// TIA Portal V20 export
// export: Created 2025-12-01T14:57:12.0152135Z, ExportSetting None, DisplayName Totally Integrated Automation Portal, DisplayVersion V20 Update 3, DisplayName TIA Portal Openness, DisplayVersion V20 Update 3, DisplayName TIA Portal Version Control Interface, DisplayVersion V20 Update 3, DisplayName STEP 7 Professional, DisplayVersion V20 Update 3, DisplayName STEP 7 Safety, DisplayVersion V20 Update 2, DisplayName WinCC Basic/Comfort/Advanced, DisplayVersion V20 Update 3, DisplayName WinCC Professional, DisplayVersion V20 Update 3, DisplayName WinCC Unified, DisplayVersion V20 Update 3
FUNCTION "FC814_EventosRec_Reset" : Void   // FC814, LAD
{ S7_Optimized_Access := 'FALSE' }
// stored: AutoNumber false, SetENOAutomatically false
   VAR_INPUT
      NumJdT : UInt;   // Numero de JdT recibido el Evento
   END_VAR
   VAR_IN_OUT
      P_Eventos : DWord;   // Puntero al DB de Eventos Recibidos
   END_VAR
   VAR_TEMP
      VarEmisionEvento : Struct
         P_Eventos : DWord;
         DBEventos : Word;
         NumDBEventos : UInt;
         MaxBytes : UInt;
         NumBytes : UInt;
         Valor : UDInt;
         Offset : UInt;
      END_STRUCT;
      DBEventosRec : Word;   // DB de Eventos Recibidos
      VarTempReset : Struct
         Mesa : UInt;
         Mckey : UDInt;
         NumeroUT : UInt;
      END_STRUCT;
      AtributosDeReset : Struct
         Tipo : DWord;
         Operacion : DWord;
         Numero : UDInt;
      END_STRUCT;
      Evento : DWord;   // Etiqueta - Evento
      Atributo : DWord;   // Etiqueta - Atributo
      EtiquetaAtributo : DWord;   // Etiqueta - Conversion de Atributo
      NumeroEvento : UInt;   // Numero de Evento
      NumeroAtributo : UInt;   // Numero de Atributo
      Indice : UInt;
      Leido : UInt;
      OffsetInicial : UInt;
      ValorDeAtributo : UDInt;   // Valor del Atributo
      ReturnValor : Int;
      Cero : Byte;
   END_VAR
BEGIN

NETWORK
TITLE = Inicializar
///////////////////////////////////////////////////////////////////////////////////////////
///////////////////////////////////////////////////////////////////////////////////////////
///////////////////////////////////////////////////////////////////////////////////////////
/// Datos del DB de Recepcion de los Eventos
      L     "JDT1_NDB_EventosRec";  // Cogemos el DB de Eventos Recibidos
      T     #DBEventosRec;
      L     "JDT1_NDB_EventosEmi";
      T     #VarEmisionEvento.DBEventos;
      T     #VarEmisionEvento.NumDBEventos;
      L     "JDT1_MaxBytes";
      T     #VarEmisionEvento.MaxBytes;

/// --- Comprobar que JDT a enviado el Evento

      L     #NumJdT;
      L     2;
      <>I;
      JC    NoRecibido_JdT02;

      L     "JDT2_NDB_EventosRec";  // Cogemos el DB de Eventos Recibidos
      T     #DBEventosRec;
      L     "JDT2_NDB_EventosEmi";
      T     #VarEmisionEvento.DBEventos;
      T     #VarEmisionEvento.NumDBEventos;
      L     "JDT2_MaxBytes";
      T     #VarEmisionEvento.MaxBytes;

NoRecibido_JdT02:NOP   0;



NETWORK
TITLE = Distribucion de los Eventos (LIsta del DB de Conversion)
/////////////////////////////////////////////////////////////////////////
/////////////////////////////////////////////////////////////////////////
/////////////////////////////////////////////////////////////////////////
// Hay que recoger el Evento, para despues repartir
// Despues '{' va el tipo de eventos (2 Bytes)
      L     #P_Eventos;  // Recogo por donde va empieza el evento
      LAR2;  // del Quimarox

      OPN   DB [#DBEventosRec];
      L     DBD [AR2, P#0.0];  // Recogo el tipo de Evento (4 Caracteres)
      T     #Evento;


/////////////////////////////////////////////////////////////////////////
/////////////////////////////////////////////////////////////////////////
/////////////////////////////////////////////////////////////////////////
// Buscar numero de evento
      L     1;
      T     #NumeroEvento;
BucleDeBusqueda_NumeroDeEvento:NOP   0;

// -- Se ha encontrado el Evento Recibido
      L     "DB870_ConversorEventos".EventosRecibidos[#NumeroEvento];
      L     #Evento;
      ==D;
      JC    Encontrado_NumeroDeEvento;

// -- Final de la lista de Eventos Recibidos - No Encontrado
      L     "DB870_ConversorEventos".EventosRecibidos[#NumeroEvento];
      L     0;
      ==D;
      JC    NoEncontrado_NumeroDeEvento;

// --- Maximo del Array de la Lista de Eventos Recibidos - No Encontrado
      L     #NumeroEvento;
      L     "CTE_MaxArrayConversion";
      >=I;
      JC    NoEncontrado_NumeroDeEvento;

// --- Continuar la Busqueda
      L     #NumeroEvento;
      L     1;
      +I;
      T     #NumeroEvento;
      JU    BucleDeBusqueda_NumeroDeEvento;


/////////////////////////////////////////////////////////////////////////
// No es ninguno de los eventos previstos, se pasa a buscar el siguiente
NoEncontrado_NumeroDeEvento:NOP   0;
      TAR2;  // Devuelve por donde va empieza el evento
      T     #P_Eventos;  // del Quimarox
      JU    Final_ListaEventos;



NETWORK
TITLE = ----
/////////////////////////////////////////////////////////////////////////
/////////////////////////////////////////////////////////////////////////
/////////////////////////////////////////////////////////////////////////
// Distribuir dependiendo del Resultado de la Busqueda del Evento Recibido
// Para recoger los Atributos
Encontrado_NumeroDeEvento:NOP   0;
      L     #NumeroEvento;
      JL    NoExiste_NumeroDeEvento;

      JU    NoExiste_NumeroDeEvento;
      JU    NoExiste_NumeroDeEvento;  // Evento (01) - CREA
      JU    NoExiste_NumeroDeEvento;  // Evento (02) - RUTA
      JU    NoExiste_NumeroDeEvento;  // Evento (03) - DRUT
      JU    NoExiste_NumeroDeEvento;  // Evento (04) - RETI
      JU    NoExiste_NumeroDeEvento;  // Evento (05) - BORR
      JU    NoExiste_NumeroDeEvento;  // Evento (06) - DATA
      JU    NoExiste_NumeroDeEvento;  // Evento (07) - ?UT?
      JU    NoExiste_NumeroDeEvento;  // Evento (08) - MOVE
      JU    NoExiste_NumeroDeEvento;  // Evento (09) - DEMB

      JU    NoExiste_NumeroDeEvento;  // Evento (10) - CSTA
      JU    NoExiste_NumeroDeEvento;  // Evento (11) - DIDO

      JU    NoExiste_NumeroDeEvento;  // Evento (12) - ORDE
      JU    NoExiste_NumeroDeEvento;  // Evento (13) - BOET
      JU    NoExiste_NumeroDeEvento;  // Evento (14) - BOBD
      JU    NoExiste_NumeroDeEvento;  // Evento (15) - RUET
      JU    NoExiste_NumeroDeEvento;  // Evento (16) - RUES
      JU    NoExiste_NumeroDeEvento;  // Evento (17) - INIR
      JU    NoExiste_NumeroDeEvento;  // Evento (18) - ?ST?

      JU    NoExiste_NumeroDeEvento;  // Evento (19) - QCRE
      JU    NoExiste_NumeroDeEvento;  // Evento (20) - QPR?

      JU    Atributos_EventosDeReset;  // Evento (21) - CHEA

/////////////////////////////////////////////////////////////////////////
NoExiste_NumeroDeEvento:NOP   0;
      TAR2;  // Devuelve por donde va empieza el evento
      T     #P_Eventos;  // del Router
      JU    Final_ListaEventos;



NETWORK
TITLE = ////////////////////////////////////////////////////////////////////////////////////////////////////////////

NETWORK
TITLE = Analizar la lista de los Atributos del Reset
Atributos_EventosDeReset:NOP   0;

/////////////////////////////////////////////////////////////////////////
/////////////////////////////////////////////////////////////////////////
/////////////////////////////////////////////////////////////////////////
// Inicializa variables de los Atributos de Quimarox
      L     0;
      T     #Cero;

      CALL  FILL
      ( BVAL    := #Cero,
        RET_VAL := #ReturnValor,
        BLK     := #AtributosDeReset
      );  // Inicializa Atributos



NETWORK
TITLE = ----
/////////////////////////////////////////////////////////////////////////
/////////////////////////////////////////////////////////////////////////
// Buscando Atributos o Final del Evento
      +AR2  P#4.0;  // Prepara Puntero para ver los atributos

InicioBucleAtributos_EventosDeReset:NOP   0;
      OPN   DB [#DBEventosRec];
      L     DBB [AR2, P#0.0];
      T     #Leido;

// Inicio de atributo - Ir a tratar los atributos
      L     #Leido;
      L     '[';  // '[' - Inicio de Atributo
      ==I;  // Atributo del Evento
      JC    EncontradoAtributos_EventosDeReset;

// Fin del Evento
      L     #Leido;
      L     '}';  // '}' - Fin del Evento
      ==I;  // Se acabo el evento
      JC    FinalAtributos_EventosDeReset;


// Sin Mensaje
      L     #Leido;
      L     0;  // No hay mas Mensaje
      ==I;  // Se acabo el evento
      JC    FinalAtributos_EventosDeReset;

      +AR2  P#1.0;  // Seguir buscado atributo
      JU    InicioBucleAtributos_EventosDeReset;


/////////////////////////////////////////////////////////////////////////
/////////////////////////////////////////////////////////////////////////
// Se acaba el Evento - Ir a guardar datos del Evento
FinalAtributos_EventosDeReset:NOP   0;
      TAR2;
      T     #P_Eventos;  // Guardo Por donde voy en la lista de eventos
      JU    GuardarDatos_EventosRecibidos;



NETWORK
TITLE = Distribucion de los Atributos del Quimarox (LIsta del DB de Conversion)
EncontradoAtributos_EventosDeReset:NOP   0;

/////////////////////////////////////////////////////////////////////////
/////////////////////////////////////////////////////////////////////////
/////////////////////////////////////////////////////////////////////////
/////////////////////////////////////////////////////////////////////////
// Mirar que Atributo del Evento  es ?
      +AR2  P#1.0;
      OPN   DB [#DBEventosRec];
      L     DBD [AR2, P#0.0];  // Atributo - 4 Caracteres
      T     #Atributo;

/////////////////////////////////////////////////////////////////////////
/////////////////////////////////////////////////////////////////////////
/////////////////////////////////////////////////////////////////////////
// Buscar numero de Atributo
      L     1;
      T     #NumeroAtributo;
BucleDeBusqueda_NumeroDeAtributoDeReset:NOP   0;

// -- Se ha encontrado el Atributo Recibido
      L     "DB870_ConversorEventos".AtributosRecibidosDeReset[#NumeroAtributo];
      L     #Atributo;
      ==D;
      JC    Encontrado_NumeroDeAtributoDeReset;

// -- Final de la lista de Atributo Recibidos - No Encontrado
      L     "DB870_ConversorEventos".AtributosRecibidosDeReset[#NumeroAtributo];
      L     0;
      ==D;
      JC    InicioBucleAtributos_EventosDeReset;

// --- Maximo del Array de la Lista de Atributo Recibidos - No Encontrado
      L     #NumeroAtributo;
      L     "CTE_MaxArrayConversion";
      >=I;
      JC    InicioBucleAtributos_EventosDeReset;


// --- Continuar la Busqueda
      L     #NumeroAtributo;
      L     1;
      +I;
      T     #NumeroAtributo;
      JU    BucleDeBusqueda_NumeroDeAtributoDeReset;



NETWORK
TITLE = ----
/////////////////////////////////////////////////////////////////////////
/////////////////////////////////////////////////////////////////////////
/////////////////////////////////////////////////////////////////////////
// Distribuir dependiendo del Resultado de la Busqueda de Atributo Recibido
Encontrado_NumeroDeAtributoDeReset:NOP   0;
      L     #NumeroAtributo;
      JL    NoExiste_NumeroDeAtibutoDeReset;

      JU    NoExiste_NumeroDeAtibutoDeReset;
      JU    AtributoDeReset_TIPO;  // Atributo (01) - TIPO
      JU    AtributoDeReset_NUME;  // Atributo (02) - NUME
      JU    AtributoDeReset_OPER;  // Atributo (03) - OPER


/////////////////////////////////////////////////////////////////////////
NoExiste_NumeroDeAtibutoDeReset:NOP   0;
      JU    InicioBucleAtributos_EventosDeReset;



NETWORK
TITLE = ---- ---- Recoger el Atributo de Quimarox - TIPO
/////////////////////////////////////////////////////////////////////////
/////////////////////////////////////////////////////////////////////////
/////////////////////////////////////////////////////////////////////////
AtributoDeReset_TIPO:NOP   0;
      +AR2  P#5.0;
      TAR2;
      T     #P_Eventos;

// Obtener el Valor del Atributo
      OPN   DB [#DBEventosRec];
      L     DBD [AR2, P#0.0];
      T     #AtributosDeReset.Tipo;

// Continuo con el Evento
      L     #P_Eventos;
      LAR2;
      +AR2  P#4.0;
      JU    InicioBucleAtributos_EventosDeReset;



NETWORK
TITLE = ---- ---- Recoger el Atributo de Quimarox - NUME
/////////////////////////////////////////////////////////////////////////
/////////////////////////////////////////////////////////////////////////
/////////////////////////////////////////////////////////////////////////
AtributoDeReset_NUME:NOP   0;
      +AR2  P#5.0;
      TAR2;
      T     #P_Eventos;
      SRD   3;
      T     #OffsetInicial;

// Obtener el Valor del Atributo
      CALL  "FC892_Obtener_ValorDelAtributo"
      ( DB_String := #DBEventosRec,
        OffsetIni := #OffsetInicial,
        Valor     := #ValorDeAtributo
      );

      L     #ValorDeAtributo;  // Lo guardo
      T     #AtributosDeReset.Numero;

// Continuo con el Evento
      L     #P_Eventos;
      LAR2;
      JU    InicioBucleAtributos_EventosDeReset;



NETWORK
TITLE = ---- ---- Recoger el Atributo de Quimarox - OPER
/////////////////////////////////////////////////////////////////////////
/////////////////////////////////////////////////////////////////////////
/////////////////////////////////////////////////////////////////////////
AtributoDeReset_OPER:NOP   0;
      +AR2  P#5.0;
      TAR2;
      T     #P_Eventos;

// Obtener el Valor del Atributo
      OPN   DB [#DBEventosRec];
      L     DBD [AR2, P#0.0];
      T     #AtributosDeReset.Operacion;

// Continuo con el Evento
      L     #P_Eventos;
      LAR2;
      +AR2  P#4.0;
      JU    InicioBucleAtributos_EventosDeReset;



NETWORK
TITLE = ////////////////////////////////////////////////////////////////////////////////////////////////////////////

NETWORK
TITLE = Distribucion para Guardar Datos del Evento Recibido (LIsta del DB de Conversion) ///////
/////////////////////////////////////////////////////////////////////////
/////////////////////////////////////////////////////////////////////////
/////////////////////////////////////////////////////////////////////////
GuardarDatos_EventosRecibidos:NOP   0;
      TAR2;
      T     #P_Eventos;  // Guardo Por donde voy en la lista de eventos

      L     #NumeroEvento;
      JL    NoExiste_GuardarDatos_Eventos;

      JU    NoExiste_GuardarDatos_Eventos;
      JU    NoExiste_GuardarDatos_Eventos;  // Evento (01) - CREA
      JU    NoExiste_GuardarDatos_Eventos;  // Evento (02) - RUTA
      JU    NoExiste_GuardarDatos_Eventos;  // Evento (03) - DRUT
      JU    NoExiste_GuardarDatos_Eventos;  // Evento (04) - RETI
      JU    NoExiste_GuardarDatos_Eventos;  // Evento (05) - BORR
      JU    NoExiste_GuardarDatos_Eventos;  // Evento (06) - DATA
      JU    NoExiste_GuardarDatos_Eventos;  // Evento (07) - ?UT?
      JU    NoExiste_GuardarDatos_Eventos;  // Evento (08) - MOVE
      JU    NoExiste_GuardarDatos_Eventos;  // Evento (09) - DEMB
      JU    NoExiste_GuardarDatos_Eventos;  // Evento (10) - CSTA
      JU    NoExiste_GuardarDatos_Eventos;  // Evento (11) - DIDO
      JU    NoExiste_GuardarDatos_Eventos;  // Evento (12) - ORDE
      JU    NoExiste_GuardarDatos_Eventos;  // Evento (13) - BOET
      JU    NoExiste_GuardarDatos_Eventos;  // Evento (14) - BOBD
      JU    NoExiste_GuardarDatos_Eventos;  // Evento (15) - RUET
      JU    NoExiste_GuardarDatos_Eventos;  // Evento (16) - RUES
      JU    NoExiste_GuardarDatos_Eventos;  // Evento (17) - INIR
      JU    NoExiste_GuardarDatos_Eventos;  // Evento (18) - ?ST?

      JU    NoExiste_GuardarDatos_Eventos;  // Evento (19) - QCRE
      JU    NoExiste_GuardarDatos_Eventos;  // Evento (20) - QPR?

      JU    GuardarDatos_EventoRecibido_CHEQ;  // Evento (21) - CHEQ


/////////////////////////////////////////////////////////////////////////
NoExiste_GuardarDatos_Eventos:NOP   0;
      JU    Final_ListaEventos;



NETWORK
TITLE = ////////////////////////////////////////////////////////////////////////////////////////////////////////////

NETWORK
TITLE = Evento CHEQ - Peticion de Datos para el Reset
GuardarDatos_EventoRecibido_CHEQ:NOP   0;

/////////////////////////////////////////////////////////////////////////
/////////////////////////////////////////////////////////////////////////
/////////////////////////////////////////////////////////////////////////
// --- Guardar Datos del Evento Recibido


/////////////////////////////////////////////////////////////////////////
/////////////////////////////////////////////////////////////////////////
/////////////////////////////////////////////////////////////////////////
/// --- Distribuir dependiendo del Tipo
      SET;  /// --- TIPO >>> Mesa
      L     #AtributosDeReset.Tipo;
      L     'MESA';
      ==I;
      JC    GuardarDatosMesa_EventoRecibido_CHEQ;

      SET;  /// --- TIPO >>> Mckey
      L     #AtributosDeReset.Tipo;
      L     'MCKY';
      ==I;
      JC    GuardarDatosMckey_EventoRecibido_CHEQ;


/// --- No Existe el Tipo
      JU    Final_EventoRecibido_CHEQ;



NETWORK
TITLE = ---- Guardar Datos de Peticion de Datos de Mesa
GuardarDatosMesa_EventoRecibido_CHEQ:NOP   0;

/////////////////////////////////////////////////////////////////////////
/////////////////////////////////////////////////////////////////////////
/////////////////////////////////////////////////////////////////////////
      L     #AtributosDeReset.Numero;
      L     "CTE_OffsetMesa";
      -I;
      T     #VarTempReset.Mesa;

// --- Control de la Mesa Recibida
      L     #VarTempReset.Mesa;  // Comprobar el numero de mesa
      L     1;  // No menor de 1
      <I;  // No es correcto
      JC    Final_EventoRecibido_CHEQ;
      L     #VarTempReset.Mesa;
      L     "CTE_MaxMesas";  // No mayor que el parametro
      >I;  // No es correcto
      JC    Final_EventoRecibido_CHEQ;


// --- Distribucion segun Operacion
      SET;  /// --- OPER >>> Ocupacion
      L     #AtributosDeReset.Operacion;
      L     'OCUP';
      ==I;
      JC    OperacionMesa_Ocupacion_EventoRecibido_CHEQ;

      SET;  /// --- OPER >>> Ocupacion
      L     #AtributosDeReset.Operacion;
      L     'MCKY';
      ==I;
      JC    OperacionMesa_Mckey_EventoRecibido_CHEQ;

      SET;  /// ---TODO >>> TODOS
      L     #AtributosDeReset.Operacion;
      L     'TODO';
      ==I;
      JC    OperacionMesa_Todas_EventoRecibido_CHEQ;


/////////////////////////////////////////////////////////////////////////
/////////////////////////////////////////////////////////////////////////
/////////////////////////////////////////////////////////////////////////
// --- Final
      JU    Final_EventoRecibido_CHEQ;



NETWORK
TITLE = ---- >>>> Operacion de Ocupacion
/////////////////////////////////////////////////////////////////////////
/////////////////////////////////////////////////////////////////////////
/////////////////////////////////////////////////////////////////////////
// --- Operacion Ocupacion de la Mesa
OperacionMesa_Ocupacion_EventoRecibido_CHEQ:NOP   0;
      SET;
      S     "DB831_Mesas".Mesas[#VarTempReset.Mesa].EventosInformarJdT.OcupacionDeMesa;

      JU    Final_EventoRecibido_CHEQ;



NETWORK
TITLE = ---- >>>> Operacion de Mckeys
/////////////////////////////////////////////////////////////////////////
/////////////////////////////////////////////////////////////////////////
/////////////////////////////////////////////////////////////////////////
// --- Operacion Mckey de la Mesa
OperacionMesa_Mckey_EventoRecibido_CHEQ:NOP   0;
      SET;
      S     "DB831_Mesas".Mesas[#VarTempReset.Mesa].EventosInformarJdT.MckeysEnMesa;

      JU    Final_EventoRecibido_CHEQ;



NETWORK
TITLE = ---- >>>> Todas las Operaciones - Ocupacion, Mckeys
/////////////////////////////////////////////////////////////////////////
/////////////////////////////////////////////////////////////////////////
/////////////////////////////////////////////////////////////////////////
// --- Todas las Operaciones de la Mesa
OperacionMesa_Todas_EventoRecibido_CHEQ:NOP   0;
      SET;
      S     "DB831_Mesas".Mesas[#VarTempReset.Mesa].EventosInformarJdT.TodoDeMesa;

      JU    Final_EventoRecibido_CHEQ;



NETWORK
TITLE = ---- Guardar Datos de Peticion de Datos de Mckey
GuardarDatosMckey_EventoRecibido_CHEQ:NOP   0;

/////////////////////////////////////////////////////////////////////////
/////////////////////////////////////////////////////////////////////////
/////////////////////////////////////////////////////////////////////////
      L     #AtributosDeReset.Numero;
      T     #VarTempReset.Mckey;

// --- Control del Mckey es correcto
      L     #VarTempReset.Mckey;  // Se ha recibido Mckey = 0
      L     0;
      ==D;
      JC    Final_EventoRecibido_CHEQ;

// --- Control del Mckey Existe
      CALL  "FC720_BuscarUT_EnMesa"
      ( Mckey      := #VarTempReset.Mckey,
        MesaActual := 0,
        NumeroUT   := #VarTempReset.NumeroUT
      );

      SET;  // Existe Mckey ?
      L     #VarTempReset.NumeroUT;
      L     0;
      ==I;
      JC    NoExisteMckey_EventoRecibido_CHEQ;
      JU    ExisteMckey_EventoRecibido_CHEQ;



NETWORK
TITLE = ---- >>>> Existe Mckey
/////////////////////////////////////////////////////////////////////////
/////////////////////////////////////////////////////////////////////////
/////////////////////////////////////////////////////////////////////////
// --- Existe Mckey
ExisteMckey_EventoRecibido_CHEQ:NOP   0;
      SET;
      S     "DB812_UTs_Control".UT[#VarTempReset.NumeroUT].EventosInformarJdT.ChequeoDelReset;

      JU    Final_EventoRecibido_CHEQ;



NETWORK
TITLE = ---- >>>> No Existe Mckey
/////////////////////////////////////////////////////////////////////////
/////////////////////////////////////////////////////////////////////////
/////////////////////////////////////////////////////////////////////////
// --- No Existe Mckey
NoExisteMckey_EventoRecibido_CHEQ:NOP   0;


////////////////////////////////////////////////////////////////////////////////
////////////////////////////////////////////////////////////////////////////////
////////////////////////////////////////////////////////////////////////////////
// Inicializo el Numero de Bytes y el puntero del DB Eventos Generados

      L     0;
      T     #VarEmisionEvento.NumBytes;  // Inicializo el numero de Bytes
      LAR2;  // Inicializo el puntero de Eventos Generados

////////////////////////////////////////////////////////////////////////////////
// Calcula el tamaño de bytes que hay en el DB Eventos Generados
InicioBucleBusquedaFin_BufferEventos:NOP   0;
      OPN   DB [#VarEmisionEvento.DBEventos];
      L     DBB [AR2, P#0.0];
      L     0;
      ==I;
      JC    FinBucleBusquedaFin_BufferEventos;  // Buscamos el final del DB = 0

      +AR2  P#1.0;
      JU    InicioBucleBusquedaFin_BufferEventos;

FinBucleBusquedaFin_BufferEventos:NOP   0;
      TAR2;  // Guardo el puntero
      T     #P_Eventos;  // Sacamos el NumBytes Escritos
      SRD   3;
      T     #VarEmisionEvento.NumBytes;

////////////////////////////////////////////////////////////////////////////////
// Comprobamos si hay sitio para mas Eventos >>>> Siempre hay Sitio Por Narices


////////////////////////////////////////////////////////////////////////////////
////////////////////////////////////////////////////////////////////////////////
////////////////////////////////////////////////////////////////////////////////
// -- Formateo del Evento CHE! - Datos UT En Reset
      L     #VarEmisionEvento.P_Eventos;
      LAR2;  // Puntero al DB de Eventos Generados

      TAR2;  // Mirar si es el primer evento de la lista
      L     0;
      ==I;
      JC    InicioBuffer_CHE_EventosUT;  // Es el primero

      OPN   DB [#VarEmisionEvento.DBEventos];  // Hay que añadir si no es el primer evento
      L     ',';  // Separador entre eventos ','
      T     DBB [AR2, P#0.0];
      +AR2  P#1.0;

InicioBuffer_CHE_EventosUT:NOP   0;
      OPN   DB [#VarEmisionEvento.DBEventos];  // DB de Eventos Generados (A Emitir)
      L     '{';  // Inicio de Evento '{'
      T     DBB [AR2, P#0.0];
      +AR2  P#1.0;

      L     'CHE!';  // Evento 'DAT?'
      T     DBD [AR2, P#0.0];
      +AR2  P#4.0;


////////////////////////////////////////////////////////////////////////////////
      OPN   DB [#VarEmisionEvento.DBEventos];
      L     '[';  // Evento - Atributo TIPO '[TIPO]'
      T     DBB [AR2, P#0.0];
      L     'TIPO';
      T     DBD [AR2, P#1.0];
      L     ']';
      T     DBB [AR2, P#5.0];
      +AR2  P#6.0;

      L     'MCKY';
      T     DBD [AR2, P#0.0];
      +AR2  P#4.0;


////////////////////////////////////////////////////////////////////////////////
      OPN   DB [#VarEmisionEvento.DBEventos];
      L     '[';  // Evento - Atributo Mckey '[NUME]'
      T     DBB [AR2, P#0.0];
      L     'NUME';
      T     DBD [AR2, P#1.0];
      L     ']';
      T     DBB [AR2, P#5.0];
      +AR2  P#6.0;

      L     #VarTempReset.Mckey;
      T     #VarEmisionEvento.Valor;

// --- Convertir Valor a ASCII - Mckey
      TAR2;
      SRD   3;
      T     #VarEmisionEvento.NumBytes;  // Miro que offset tiene la String

      CALL  "FC893_Obtener_StringDelAtributo"
      ( DB_String := #VarEmisionEvento.NumDBEventos,
        OffsetIni := #VarEmisionEvento.NumBytes,
        Valor     := #VarEmisionEvento.Valor,
        OffsetFin := #VarEmisionEvento.Offset
      );  // Llamo a ObtenerStrinAtributo

      L     #VarEmisionEvento.Offset;
      SLD   3;
      LAR2;  // Recupero que offset tiene la String

// --- Ya esta convertido el Valor a ASCI - Fin Mckey


////////////////////////////////////////////////////////////////////////////////
      OPN   DB [#VarEmisionEvento.DBEventos];
      L     '[';  // Evento - Atributo Resultado '[RESU]'
      T     DBB [AR2, P#0.0];
      L     'RESU';
      T     DBD [AR2, P#1.0];
      L     ']';
      T     DBB [AR2, P#5.0];
      +AR2  P#6.0;

      L     'FALS';
      T     DBD [AR2, P#0.0];
      L     'E';
      T     DBB [AR2, P#4.0];
      +AR2  P#5.0;


////////////////////////////////////////////////////////////////////////////////
// --- Final del Formato del Evento ---

      OPN   DB [#VarEmisionEvento.DBEventos];  // DB de Eventos Generados (A Emitir)
      L     '}';  // Fin de Evento '}'
      T     DBB [AR2, P#0.0];
      +AR2  P#1.0;

      JU    Final_EventoRecibido_CHEQ;



NETWORK
TITLE = ---- Final
///////////////////////////////////////////////////////////////////////////////
///////////////////////////////////////////////////////////////////////////////
///////////////////////////////////////////////////////////////////////////////
// --- Se acabo el evento
Final_EventoRecibido_CHEQ:NOP   0;
      L     #P_Eventos;  // Recupero por donde voy en la lista de eventos
      LAR2;  // Regreso a buscar el siguiente evento
      JU    Final_ListaEventos;



NETWORK
TITLE = Final de la Lista de Eventos
///////////////////////////////////////////////////////////////////////////////////////////
///////////////////////////////////////////////////////////////////////////////////////////
///////////////////////////////////////////////////////////////////////////////////////////
/// Final de la Recepcion de la Lista de Eventos
Final_ListaEventos:NOP   0;


END_FUNCTION
